// TwinCAT 3 PLC project Dimmer
// ProgramVersion: 3.1.4023.0
// libraries:
//   Tc2_Standard, * (Beckhoff Automation GmbH)
//   Tc2_System, * (Beckhoff Automation GmbH)
//   Tc3_IotCommunicator, * (Beckhoff Automation GmbH)
//   Tc3_Module, * (Beckhoff Automation GmbH)
// project tree:
//   DUTs/ ST_ProcessData.TcDUT
//   GVLs/ gvl_IO.TcGVL
//   / PlcTask.TcTTO
//   POUs/ FB_Dimmer.TcPOU, FB_SectorUpdate.TcPOU, FB_TriStableSwitch.TcPOU, FB_TriStableSwitchHisteresis.TcPOU, MAIN.TcPOU
// real-time tasks:
//   TASK PlcTask: cycle T#10ms, priority 20, ADS port 350

CONFIGURATION Dimmer
    RESOURCE PLC ON TwinCAT3
        TASK PlcTask(INTERVAL := T#10ms, PRIORITY := 20);
        PROGRAM MAIN WITH PlcTask : MAIN;
    END_RESOURCE
END_CONFIGURATION

// ---- DUTs/ST_ProcessData.TcDUT
TYPE ST_ProcessData :
STRUCT 
	{attribute 'iot.DisplayName' := 'Chłodzenie'}
	bCoolingInfo : BOOL;
	{attribute 'iot.DisplayName' := 'Grzanie'}
	bHeatingInfo : BOOL;
	
	
	
	{attribute 'iot.DisplayName' := 'Power'} 
	bPower : BOOL;

	{attribute 'iot.DisplayName' := 'Light Intensity'} 
	{attribute 'iot.ReadOnly' := 'true'} 
	{attribute 'iot.MinValue' := '0'} 
	{attribute 'iot.MaxValue' := '255'} 
	iLightIntensity : INT; 

END_STRUCT 
END_TYPE

// ---- GVLs/gvl_IO.TcGVL
{attribute 'qualified_only'}
VAR_GLOBAL
	//INPUTS
	bButton1	AT%I*	:BOOL;	//bistabilny
	bButton2	AT%I*	:BOOL;	//bistabilny
	bButton3	AT%I*	:BOOL;	//monostabilny
	bButton4	AT%I*	:BOOL;	//monostabilny
	
	iAnalog1	AT%I*	:INT;	//potencjometr 1
	iAnalog2	AT%I*	:INT;	//potencjometr 2
	
	//OUTPUTS
	
	bOutput1	AT%Q*	:BOOL;	//wyjście 1
	bOutput2	AT%Q*	:BOOL;	//wyjście 2
END_VAR

// ---- POUs/MAIN.TcPOU
PROGRAM MAIN
VAR
	(*
	tssAnalog		:FB_TriStableSwitch;
	byOswietlenie	:BYTE:=0;
	fbDimmer1		:FB_Dimmer;
	fbIoT 			: FB_IotCommunicator := ( 
										sHostName := '192.168.1.122', 
										nPort := 1883, 
										sMainTopic := 'Dimmer',
										sDeviceName := 'BeckhoffSzkolenie');
										
	stData: ST_ProcessData;     // Values to send
	tonTimer : TON;             // Timer to send data
	*)
	
	tsshTermostat		:FB_TriStableSwitchHisteresis;
END_VAR

(*
//Tri-Stable Switch; Ogrzewanie/Chłodzenie
tssAnalog(iAnalog:=gvl_IO.iAnalog1, bCooling=>gvl_IO.bOutput1, bHeating=>gvl_IO.bOutput2);
stData.bCoolingInfo:=tssAnalog.bCooling;
stData.bHeatingInfo:=tssAnalog.bHeating;

// Dimmer
fbDimmer1(bEnable:=stData.bPower, bControl:=gvl_IO.bButton3, tTimeOutLimit:=T#1S, bySignal=>byOswietlenie);
stData.iLightIntensity:=BYTE_TO_INT(fbDimmer1.bySignal);

//Komunikacja IoT
fbIoT.Execute(TRUE); //keep communication alive 
tonTimer(IN := NOT tonTimer.Q, PT := T#500MS);

IF fbIoT.bConnected AND tonTimer.Q THEN		//przesył danych do Brokera
    fbIoT.SendData(ADR(stData), SIZEOF(stData));
END_IF

IF fbIoT.fbCommand.bAvailable THEN	//nadpisanie danych do sterownika
    IF fbIoT.fbCommand.sVarName = 'bPower' THEN
        fbIoT.fbCommand.GetValue(ADR(stData.bPower), SIZEOF(stData.bPower), E_IotCommunicatorDatatype.type_BOOL);
    END_IF
    fbIoT.fbCommand.Remove();
END_IF

//przykład wiadomości
//fbIoT.SendMessage('This is a test alarm message!');
*)

tsshTermostat(iAnalogInput:=gvl_IO.iAnalog1, bHeating=>gvl_IO.bOutput2, bCooling=>gvl_IO.bOutput1);

END_PROGRAM

// ---- POUs/FB_TriStableSwitchHisteresis.TcPOU
(*
Blok włącza ogrzewaniu, chłodzenie lub nic nie robi w zależności od temperatury i historii układu.
Temperaturę symuluje nastawa potencjometru analogowego.
Traktuje się go jako switch tristabilny z podwójną histerezą pracy.

-----INPUTS-----
Jak w deklaracji poniżej.
-----OUTPUTS-----
Jak w deklaracji poniżej.

-----Uwagi-----
Brak

Wersja:
TwinCAT		3.1.4024.10
Wersja		1.0
Data		07.2020
*)
FUNCTION_BLOCK PUBLIC FB_TriStableSwitchHisteresis
VAR_INPUT
	iAnalogInput		:INT:=0;	//wejście analogowa symulujące zmianę temperatury
	
	iEnableHeating		:INT:=5;	//temperatura załączenia grzania
	iDisableHeating		:INT:=10;	//temperatura wyłączenia grzania
	iDisableCooling		:INT:=20;	//temperatura wyłączenia chłodzenia
	iEnableCooling		:INT:=25;	//temperatura włączenia chłodzenia
	
	iTempMin			:INT:=0;	//temperatura na potencjometrze w pozycji dolnej granicznej
	iTempMax			:INT:=40;	//temperatura na potencjometrze w pozycji górnej granicznej
END_VAR
VAR_OUTPUT
	bHeating		:BOOL:=FALSE;	//wyjście sterujące urządzeniem grzejącym
	bCooling		:BOOL:=FALSE;	//wyjście sterujące urządzeniem chłodzącym
END_VAR
VAR
	iTemp				:INT:=0;		//obecna temperatura
	iSectorTemp			:INT:=0;		//dobrany sektor pracy na bazie temperatury
	iCurrentSector		:INT:=0;		//obecny sektor
	iPreviousSector		:INT:=0;		//poprzedni sektor [1,2,3,4,5]
	
	suUpdate			:FB_SectorUpdate;
END_VAR

//odczyt temperatury - przeskalowanie wejścia analogowego do zadanych granic temperatury 
iTemp:=iAnalogInput*(iTempMax-iTempMin)/32676+iTempMin;

//przypisanie sektora na bazie temperatury
IF iTemp > iTempMin AND iEnableHeating > iTemp 			THEN iSectorTemp:=1; END_IF
IF iTemp > iEnableHeating AND iDisableHeating > iTemp 	THEN iSectorTemp:=2; END_IF
IF iTemp > iDisableHeating AND iDisableCooling > iTemp 	THEN iSectorTemp:=3; END_IF
IF iTemp > iDisableCooling AND iEnableCooling > iTemp 	THEN iSectorTemp:=4; END_IF
IF iTemp > iEnableCooling AND iTempMax > iTemp 			THEN iSectorTemp:=5; END_IF

CASE iSectorTemp OF
	1:	//sektor 1, w którym grzanie jest zawsze włączone
		//uaktualnienie historii układu
		suUpdate(iS:=1, iCS_IN_OUT:=iCurrentSector, iPS_IN_OUT:=iPreviousSector);
		bHeating:=TRUE;
		bCooling:=FALSE;
	2:	//sektor 2
		//uaktualnienie historii układu
		suUpdate(iS:=2, iCS_IN_OUT:=iCurrentSector, iPS_IN_OUT:=iPreviousSector);
		CASE iPreviousSector OF			//jeżeli poprzednim sektorem był
			1:
				bHeating:=TRUE;			//1, wtedy załącz grzanie
				bCooling:=FALSE;		
			3:
				bHeating:=FALSE;		//3, wtedy stan neutralny
				bCooling:=FALSE;
		END_CASE
	3:	////sektor 3, w którym grzanie i chłodzenie są wyłączone
		//uaktualnienie historii układu
		suUpdate(iS:=3, iCS_IN_OUT:=iCurrentSector, iPS_IN_OUT:=iPreviousSector);
		bHeating:=FALSE;
		bCooling:=FALSE;
	4:	//sektor 4
		//uaktualnienie historii układu
		suUpdate(iS:=4, iCS_IN_OUT:=iCurrentSector, iPS_IN_OUT:=iPreviousSector);
		CASE iPreviousSector OF			//jeżeli poprzednim sektorem był
			3:
				bHeating:=FALSE;		//3, wtedy stan neutralny
				bCooling:=FALSE;
			5:
				bHeating:=FALSE;		//5, wtedy załącz chłodzenie
				bCooling:=TRUE;
		END_CASE
	5:	//sektor 5, w którym chłodzenie jest zawsze włączone
		//uaktualnienie historii układu
		suUpdate(iS:=5, iCS_IN_OUT:=iCurrentSector, iPS_IN_OUT:=iPreviousSector);
		bHeating:=FALSE;
		bCooling:=TRUE;
END_CASE

END_FUNCTION_BLOCK

// ---- POUs/FB_SectorUpdate.TcPOU
FUNCTION_BLOCK PUBLIC FB_SectorUpdate
VAR_INPUT
	iS		:INT;	//numer sektora, z którego przyszło zapytanie
END_VAR
VAR_OUTPUT
END_VAR
VAR
END_VAR
VAR_IN_OUT
	iCS_IN_OUT	:INT;	//sektor zapisany jako obecny
	iPS_IN_OUT	:INT;	//sektor zapisany jako poprzedni
END_VAR

IF iS=iCS_IN_OUT THEN			//jeżeli sektor, z którego przyszło zapytanie jest zapisany jako obecny
	;							//nic nie rób
ELSE							//w przeciwnym wypadku		
	iPS_IN_OUT:=iCS_IN_OUT;		//zapisz sektor stary obecny jako poprzedni 
	iCS_IN_OUT:=iS;             //a ten z którego przyszło zapytanie jako obecny                      
END_IF

END_FUNCTION_BLOCK

// ---- POUs/FB_Dimmer.TcPOU
(*
Opis bloku FB_Dimmer

Blok służy do obsługi oświetlenia funkcją dimmer.
Oprócz klasycznego ON/OFF, wyjście może być sterowane płynnie w górę i w dół.
Cała kontrola odbywa się za pomocą jednego wejścia, preferowany przycisk monostabilny.

Charakterystyka pracy
Krótkie naciśnięcie powoduje gwałtowne wyłączenie/włączenie światła na wyjściu z bloku.
Przytrzymanie powoduje stopniowe rozjaśnianie i ściemnianie na przemiennie.
Po wyłączeniu oświetlenia krótkim naciśnięciem i ponownym włączeniu, powraca ono do natężenia z przed wyłączenia.

-----INPUTS-----
bEnable		:BOOL:=FALSE;		//wejście uruchamiające cały blok; TRUE - dimmer działa, FLASE - dimmer jest wyłączony
bControl	:BOOL:=FALSE;		//symulacja przycisku; TRUE - ON, FALSE  - OFF
tTimeOutLimit	:TIME:=T#1S;	//graniczny czas wciśnięcia przycisku, będący wyróżnikiem trybu pracy przycisku
	
-----OUTPUTS-----
bySignal	:BYTE:=0;	//wyjście na oświetlenie, gdzie 0-wyłączone, 255-w pełni włączone

-----Uwagi-----


Wersja:
TwinCAT 	3.1.4024.10
Ver 		1.0
Data		07.2020
*)

FUNCTION_BLOCK PUBLIC FB_Dimmer
VAR_INPUT
	bEnable		:BOOL:=FALSE;	//wejście uruchamiające cały blok; TRUE - dimmer działa, FLASE - dimmer jest wyłączony
	bControl	:BOOL:=FALSE;	//symulacja przycisku; TRUE - ON, FALSE  - OFF
	tTimeOutLimit	:TIME:=T#1S;	//graniczny czas wciśnięcia przycisku, będący wyróżnikiem trybu pracy przycisku
END_VAR
VAR_OUTPUT
	bySignal	:BYTE:=0;	//wyjście na oświetlenie, gdzie 0-wyłączone, 255-w pełni włączone
END_VAR
VAR
	bFlagON			:BOOL:=FALSE;	//zmienna określająca stan oświetlenia; TRUE-światło włączone, FALSE-światło wyłączone
	bFlagValueInMemory	:BOOL:=FALSE;	//informacja o tym, że lampa w poprzednim stanie miała określone natężenie, które zostało zapisane w pamięci
	bFlagEdge		:BOOL:=TRUE;	//zmienna określająca kierunek zmiany natężenia; TRUE-zwiększanie, FALSE-zmniejszanie
	bFlagTimeOut	:BOOL:=FALSE;	//zmienna określająca przekroczenie czasu granicznego naciśnięcia, będący wyróżnikiem trybu pracy przycisku
	bFlagShort		:BOOL:=FALSE;	//określenie czy naciśnięcie było krótkie czy długie; TRUE-krótkie, FALSE-długie
	bySignalMemory	:BYTE:=0; 		//zmienna zapamiętująca aktualny stan wyjścia
	ftrigControl	:F_TRIG;		//wykrycie zbocza malejącego na wejściu bControl
	rtrigControl	:R_TRIG;		//wykrycie zbocza rosnącego na wejściu bControl
	tonTimer		:TON;			//odmierzanie czasu wstępnego wciśnięcia przycisku
	bTimerInWork	:BOOL:=FALSE; 	//podtrzymanie timera tonTimer na czas wstępny
	tonTimerDimmerImpulse	:TON;	//timer tworzący impulsy co określony czas
	bTimerDimmerImpulse		:BOOL:=FALSE;	//podtrzymanie tonTimerDimmerImpulse, na czas wciśnięcia bControl
END_VAR

ftrigControl(CLK:=bControl);	//inicjalizacja wykrywania zbocza malejącego na zmiennej bControl
rtrigControl(CLK:=bControl);	//inicjalizacja wykrywania zbocza rosnącego na zmiennej bCOntrol
IF bEnable=TRUE THEN
	
	IF rtrigControl.Q=TRUE THEN	bTimerInWork:=TRUE;	END_IF	// start timera tonTimer następuje, gdy wykryte zostanie zbocze rosnące na bControl
	tonTimer(IN:=bTimerInWork, PT:=tTimeOutLimit);			// wyłączony zostaje on po określonym czasie tTimeOutLimit
	IF tonTimer.Q=TRUE THEN							//jeżeli timer doliczy do końca wyłącz go poprzez ustawienie flagi bTimerInWork na FALSE
		bTimerInWork:=FALSE;	
	END_IF
	IF bTimerInWork AND ftrigControl.Q = TRUE THEN	//jeżeli timer odlicza i wystąpi zbocze malejące na bControl ustaw flagę bFlagShort na TRUE
		bFlagShort:=TRUE;							//oznacza to, że wciśnięcie jest krótkie
	END_IF
	IF tonTimer.Q=TRUE AND bControl=TRUE THEN	//jeżeli odliczanie timera się zakończy, a bControl nadal jest TRUE, ustaw flagę bFlagShort na FALSE
		bFlagShort:=FALSE;						//oznacza to, że wciśnięcie jest długie
		bTimerDimmerImpulse:=TRUE;				//załączenie tonTimerDimmerImpulse
	END_IF
	
	//inicjalizacja pulsatora o okresie 10ms
	tonTimerDimmerImpulse(IN:=bTimerDimmerImpulse AND NOT tonTimerDimmerImpulse.Q, PT:=T#10MS);
	
	//jeżeli wykryto zbocze malejące na bControl i tonTimerDimmerImpulse działa, wyłącz go
	IF ftrigControl.Q=TRUE AND bTimerDimmerImpulse=TRUE THEN
		bTimerDimmerImpulse:=FALSE;
		IF bFlagEdge=TRUE THEN
			bFlagEdge:=FALSE;
		ELSE
			bFlagEdge:=TRUE;
		END_IF
	END_IF
	
	CASE bySignal OF
		0:									//przypadek, gdy światło jest wyłączone
				IF bFlagShort=TRUE THEN		//jeżeli wykryte zostało wciśnięcie krótkie
					bFlagON:=TRUE;			//ustaw flagę bFlagON na TRUE
					IF bFlagValueInMemory THEN		//jeżeli lampa została wyłączona krótko
						bySignal:=bySignalMemory;	//przywrócenie stanu lampy z przed wyłączenia
						bFlagValueInMemory:=FALSE;	//reset flagi mówiącej o zapisanej wartości wyjścia w pamięci
					ELSE
						bySignal:=255;			//w przeciwnym przypadku ustaw bySignal na 255, co oznacza pełne włączenie
					END_IF
					bFlagShort:=FALSE;		//reset flagi bFlagShort mówiący o wykonaniu czynności wywołanej krótkim wciśnięciem
				END_IF
				
				IF bTimerDimmerImpulse=TRUE THEN	//jeżeli wciśnięcie jest długie
					IF bFlagEdge=TRUE THEN			//oraz kierunek jest rosnący
						bFlagON:=TRUE;		//ustaw flagę bFlagON na TRUE; włącz lampę
						bySignal:=1;		//ustaw natężenie na minimalne =1
					END_IF
				END_IF
			
		255:								//przypadek, gdy światło jest włączone w pełni
				IF bFlagShort=TRUE THEN		//jeżeli wykryte zostało wciśnięcie krótkie
					bFlagON:=FALSE;			//ustaw flagę bFlagON na FALSE
					bySignal:=0;			//oraz ustaw bySignal na 0, co oznacza pełne wyłączenie
					bFlagShort:=FALSE;		//reset flagi bFlagShort mówiący o wykonaniu czynności wywołanej krótkim wciśnięciem
				END_IF
				
				IF  bTimerDimmerImpulse=TRUE THEN	//jeżeli wciśnięcie jest długie
					IF bFlagEdge=FALSE THEN			//oraz kierunek jest malejący
						bySignal:=254;				//ustaw natężenie na prawie maksymalne 254
					END_IF
				END_IF
		ELSE								//światło o szarym natężeniu
				IF bFlagShort=TRUE THEN		//jeżeli wykryte zostało wciśnięcie krótkie
						bySignalMemory:=bySignal;		//zapisz obecne natężenie do miennej bySignalMemory
						bFlagValueInMemory:=TRUE;		//ustawienie informacji, że wartość natężenia z przed wyłączenia czeka w pamięci
						bySignal:=0;					//ustaw nowe natężenie =0
						bFlagON:=FALSE;					//ustaw flagę bFlagON=FALSE, świadczy to o wyłączeniu lampy
						bFlagShort:=FALSE;		//reset flagi bFlagShort mówiący o wykonaniu czynności wywołanej krótkim wciśnięciem
				END_IF

				IF bTimerDimmerImpulse=TRUE THEN	//jeżeli wciśnięcie jest długie
					IF tonTimerDimmerImpulse.Q=TRUE THEN	//na każdy impuls z impulsatora
						IF bFlagEdge=TRUE THEN			//gdy kierunek jest rosnący
							bySignal:=bySignal+1;		//zwiększ natężenie o 1
						ELSE							//gdy kierunek jest malejący
							bySignal:=bySignal-1;		//zmniejsz natężenie o 1
						END_IF
					END_IF
				END_IF
	END_CASE

END_IF

END_FUNCTION_BLOCK

// ---- POUs/FB_TriStableSwitch.TcPOU
FUNCTION_BLOCK PUBLIC FB_TriStableSwitch
VAR_INPUT
	iAnalog		:INT:=0;
END_VAR
VAR_OUTPUT
	bCooling	:BOOL:=FALSE;
	bHeating	:BOOL:=FALSE;
END_VAR
VAR
	iSelector	:INT:=0;
END_VAR

iSelector:=iAnalog/10892;
CASE iSelector OF
	0:
		bCooling:=TRUE;
		bHeating:=FALSE;
	1:
		bCooling:=FALSE;
		bHeating:=FALSE;
	2:
		bCooling:=FALSE;
		bHeating:=TRUE;
END_CASE

END_FUNCTION_BLOCK
